// Simulates the heater temperature
//
FUNCTION_BLOCK FB_HeaterSimu
VAR_INPUT
END_VAR
VAR
	
	// Other members...
	Cntr:        SINT; // Counter
	Power:       SINT; // Heating power [0...100 %]
	PowerLast:   SINT; // Last heating power [0...100 %]
	Speed:       REAL; // Heating speed [+/- °C/s]
	Temperature: REAL; // Temperature [°C]
	TempTarget:  REAL; // Target temperature from the active power level [°C]
	
END_VAR

// Is restart requested ?
IF IO_Inputs.i_Restart THEN

	// Restart members
	Cntr        := 0;
	Power       := 0;
	PowerLast   := 0;
	Speed       := 0;
	Temperature := 0;
	
END_IF

// Is heater controlled to ON ?
IF IO_Inputs.i_HtrON THEN
	
	// Increase the heating power [%]
	Power := ( Power + 1 );
	
END_IF

// Is visited 100 times ?
IF Cntr = 100 THEN
	
	// Restart the visiting counter
	Cntr := 1;
	
// else, Not 100 times yet
ELSE
	
	// Increase the visiting counter
	Cntr := ( Cntr + 1 );
	RETURN;
	
END_IF

// Be sure the device movement is slow
Power := LIMIT( MAX( 0, PowerLast - 10 ), Power, MIN( 100, PowerLast + 10 ));

// Tune the power (dead time)
Power := (( Power + ( PowerLast * 2 )) / 3 );
 
// Define the final temperature based from the active power level [°C]
TempTarget := ( 10 + ( Power * 1.9 )); // 0 ...100 % => 10 ... 200 °C
  
// Define the heating speed  [+/- °C/s]
Speed := LIMIT( -2, Speed + (( TempTarget - Temperature ) / 300 ), 2 );

// Update new temperature [°C]
Temperature := LIMIT( 0, Temperature + Speed, 999 );

// Write temperature to I/O output [°C]
IO_Outputs.o_HtrTemp := Temperature;

// Save the latest power 
PowerLast := Power;
Power     := 0;

END_FUNCTION_BLOCK

(* stored: Version 1.1.0.1, ProductVersion 3.1.4022.6
   POU FB_HeaterSimu: Id {66d8a00c-59a2-48d1-bb92-9b45d33de25d}, SpecialFunc None *)
